Staubli VAL3: insertInstr.pgx

program insertInstr(InstrItem& x_sItem[])
  local num i
  local string l_sMessage
  local num l_nIndex
  local string l_sPath
  local string l_sItem
  local string l_sData
begin
  call use:setSizeList(19,0,19,11)
  call use:setView(false)
  call language2:message(l_sMessage,16)
  call use:listcreate(l_sMessage)
  // insert the action on Point
  call use:listadd(saveData:sInstrOnPoint)
  call use:listupdate(0)
  // SELECT THE ITEM
  x_sItem.sType=""
  x_sItem.sData=""
  do
    i=get()
    l_nIndex=0
    call use:listevent(i,l_nIndex,l_sItem)
  until i==255 or i==270
  //
  if l_sItem!="" and i==270
    call saveData:getPathInstr(l_sItem,l_sPath)
    events:libLoad(l_sPath)
    delay(0)
    call events:onInsert(l_sData)
    // insert the item
    x_sItem.sType=l_sItem
    x_sItem.sData=l_sData
    return
  endIf
  // NOT GOOD
  x_sItem.sType=""
  x_sItem.sData=""
  call use:nullKey(nKey)
end
